FUNCTION GetWaterDuration : TIME
VAR_INPUT
	MoistIn:REAL ;
	TempIn:REAL;
END_VAR
VAR
	rSeconds : REAL; 
    udiMs : UDINT; // milliseconds as unsigned integer
END_VAR

// Calculate duration in seconds
rSeconds := 10.0 + (TempIn - 20.0) - (MoistIn * 0.1);

// Convert to ms, then to UDINT
udiMs := LREAL_TO_UDINT(REAL_TO_LREAL(rSeconds) * 1000.0);

// Convert to TIME
GetWaterDuration := UDINT_TO_TIME(udiMs);

// Clamp between 5s and 30s
IF GetWaterDuration < T#5s THEN GetWaterDuration := T#5s; END_IF;
IF GetWaterDuration > T#30s THEN GetWaterDuration := T#30s; END_IF;

END_FUNCTION

(* stored: Version 1.1.0.1, ProductVersion 3.1.4024.15
   POU GetWaterDuration: Id {0e665143-0f50-47dc-b43f-c2460d0fd759}, SpecialFunc None *)
